FUNCTION_BLOCK FB_OffState IMPLEMENTS I_State
VAR_INPUT
END_VAR
VAR_OUTPUT
END_VAR
VAR
	pConveyorSystem : POINTER TO FB_ConveyorSystem;
END_VAR

{warning 'add property implementation'}
PROPERTY Description : STRING
GET
Description := 'Off state';
END_GET
END_PROPERTY

{warning 'add method implementation '}
METHOD DetectedPartSensor1 : BOOL
END_METHOD

{warning 'add method implementation '}
METHOD DetectedPartSensor2 : BOOL
END_METHOD

{warning 'add method implementation '}
METHOD DetectedWeightSensor : BOOL
END_METHOD

METHOD FB_init : BOOL
VAR_INPUT
	bInitRetains : BOOL; // if TRUE, the retain variables are initialized (warm start / cold start)
	bInCopyCode : BOOL;  // if TRUE, the instance afterwards gets moved into the copy code (online change
	pConveyorSystem : POINTER TO FB_ConveyorSystem;
END_VAR
THIS^.pConveyorSystem := pConveyorSystem;
END_METHOD

{warning 'add method implementation '}
METHOD PressEmergencyStop : BOOL
END_METHOD

{warning 'add method implementation '}
METHOD PressStart : BOOL
pConveyorSystem^.SetState(pConveyorSystem^.IdleState);
END_METHOD

{warning 'add method implementation '}
METHOD PressStop : BOOL
END_METHOD

{warning 'add method implementation '}
METHOD ProcessedWeight : BOOL
END_METHOD

END_FUNCTION_BLOCK

(* stored: Version 1.1.0.1, ProductVersion 3.1.4024.12
   POU FB_OffState: Id {f767024e-3326-46ec-8144-2d5eeb633a6b}, SpecialFunc None
   Property Description: Id {41ba9f15-24b3-42c8-a6e1-3fec389ccb27}
   Get Get: Id {135eb60f-2b75-4e6f-8055-29dbb2978634}
   Method DetectedPartSensor1: Id {11f4fceb-12da-47f5-9257-c9a3729acd80}
   Method DetectedPartSensor2: Id {53134cca-a2be-4e2f-99bb-9b07e0858e5f}
   Method DetectedWeightSensor: Id {5e525a8e-0377-4745-86cb-3ffa9125451d}
   Method FB_init: Id {24d0da4f-3090-44f3-8ada-5436d3af5bb0}
   Method PressEmergencyStop: Id {a4d4c721-9b82-4b5a-ae8c-1c2b86da4784}
   Method PressStart: Id {682399fa-abfd-4276-b2c8-7b4212b3f8df}
   Method PressStop: Id {32c03365-5e85-42a1-943c-17c9a0e6d9e1}
   Method ProcessedWeight: Id {6e0de949-f75b-4510-a0d3-baa50a807f2d} *)
